PROGRAM MAIN
VAR
END_VAR

// Orquestracao preenchida na Task 14.

END_PROGRAM

(* stored: Version 1.1.0.1
   POU MAIN: Id {34154070-d696-46ff-9128-cc1ffe67f4c4}, SpecialFunc None *)
